TYPE Rec_Pusher :
	STRUCT
		//Initial_Speed				:LREAL;
		//Initial_Distance			:LREAL;
		//Eject_Speed					:LREAL;
		//Eject_Distance				:LREAL;
		//Retract_Speed				:LREAL;
		//tamp_initial_speed			:LREAL;
		//tamp_final_speed			:LREAL;
		//tamp_initial_distance		:LREAL;
		//tamp_final_distance			:LREAL;
		
		Speed				:ARRAY[1..6] OF LREAL;
		Distance			:ARRAY[1..6] OF LREAL;
		retract_speed			:LREAL;
		
	END_STRUCT
END_TYPE

(* stored: Version 1.1.0.1, ProductVersion 3.1.4020.12
   DUT Rec_Pusher: Id {84aa4b80-3b97-4d1a-be08-8a9b0efe8a1f} *)
